RoboDK station: FollowCurves_Inatel.rdk

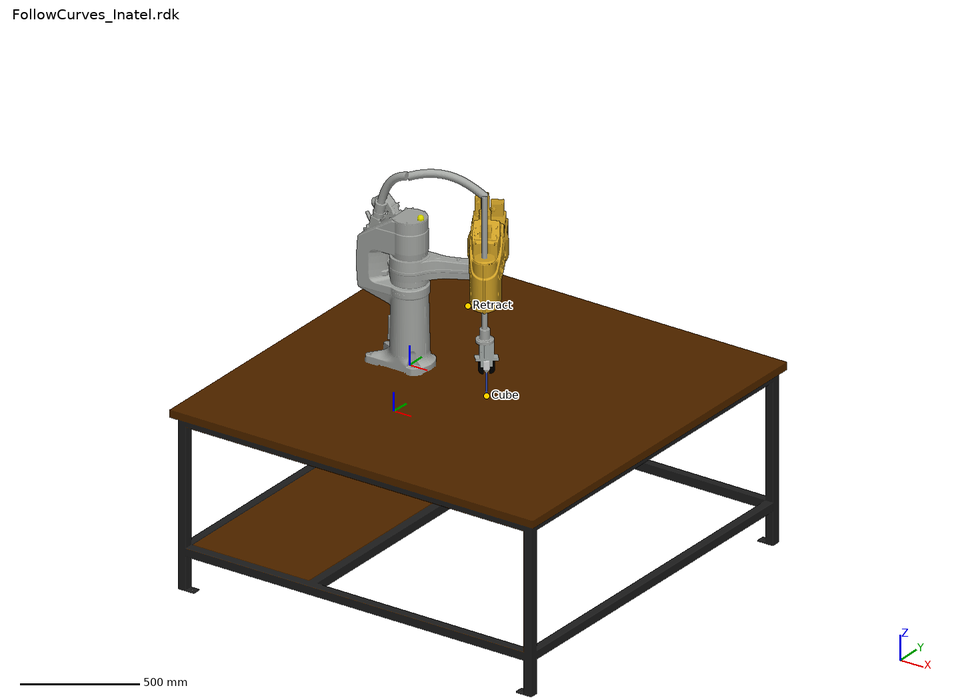
[picture v0: the station drawn from its stored meshes, robots at their saved joint values, targets as dots, program paths as lines]
Station FollowCurves_Inatel (saved by RoboDK 5.4.1). Poses are relative to the parent item; angles as X-Y-Z fixed-axis rotations.
Station parameters (name, value as stored): LIN64
  - frame World at (0, 0, 835) mm
    - robot Staubli TS60 FL 200 (model Staubli TS60 FL 400): 4 axes, payload 2 kg, reach 600 mm, repeatability 0.01 mm, weight 55 kg
        modified DH rows (alpha deg, a mm, theta deg, d mm): 0, 0, 0, 0; 0, 330, 0, 0; 0, 270, 0, 170 linear; 180, 0, 0, 0
        joint limits [-140, -150, 0, -500] to [140, 150, 200, 500]; home [0, 0, 0, 0]; saved at [27.421, -85.421, 90, 122]
      - tool GarraCompleta, TCP at (0, 0, 200) mm, size 97 x 40 x 153.1 mm, geometry from GarraCompleta.STL
        - object Suporte_e_Caneta at (4.39, 18.92, -137) mm, rotated rx 0 ry 0 rz 48 deg, size 26 x 26 x 165.9 mm, geometry from Suporte_e_Caneta.STL
      - tool TCP_Garra, TCP at (0, 17, 260) mm
    - target Retract (Cartesian target) at (-121.61, 599.78, 0) mm, rotated rx 180 ry 0 rz -180 deg; joints [108.252, -14.375, 90, 273.877] of Staubli TS60 FL 200
  - object Mesa at (350, 0, 0) mm, size 1850 x 1850 x 835 mm, geometry from Mesa.STL
  - frame AreaTrabalho at (200, -400, 835) mm
    - target Cube (Cartesian target) at (236, 340, 0) mm, rotated rx 180 ry 0 rz 180 deg; joints [22.348, -85.774, 90, 116.574] of Staubli TS60 FL 200
  - Python program dynamicTarget (listed below)

--- Python program dynamicTarget ---
from robodk.robolink import *      # RoboDK's API
from robodk.robomath import *      # Math toolbox for robots
from tkinter import *
import numpy as np
import cv2

def getElements(image):
    imgHSV = cv2.cvtColor(image, cv2.COLOR_BGR2HSV)
    lower = np.array([32, 0, 0])
    upper = np.array([145, 255, 255])
    mask = cv2.inRange(imgHSV, lower, upper)
    imgResult = cv2.bitwise_and(image, image, mask=mask)
    return imgResult

def showImages(images):
    for image in images:
        cv2.imshow('Image', image)
        cv2.waitKey(0)
        cv2.destroyAllWindows()

def getPosition():
    path = '/home/fabiofiorita/Documentos/IC-Gemeo/Localização de Objetos/DynamicTarget/bancada1.png'
    image = cv2.imread(path)
    #image = cv2.resize(image, (1200, 2000))
    maskedImage = getElements(image)

    img = maskedImage.copy()
    im_bw = cv2.cvtColor(img, cv2.COLOR_RGB2GRAY)
    #blur = cv2.GaussianBlur(im_bw, (5,5), 0)
    #im_bw = cv2.Canny(blur, 10, 90)
    contours, hierarchy = cv2.findContours(im_bw, cv2.RETR_TREE, cv2.CHAIN_APPROX_SIMPLE)
    centers = []
    for c in contours:
        M = cv2.moments(c)
        if M['m00'] != 0:
            cx = int(M['m10']/M['m00'])
            cy = int(M['m01']/M['m00'])
            cv2.drawContours(img, [c], -1, (0,255,0), 3)
            cv2.circle(img, (cx, cy), 5, (0,0,255), -1)
            cv2.putText(img, f"{cx, cy}", (cx - 20, cy - 20), cv2.FONT_HERSHEY_SIMPLEX, 0.5, (0,0,255), 2)
            centers.append((cx, cy))
    showImages([image, maskedImage, img])
    return centers

def interface():
    centers = getPosition()

    master = Tk()
    master.geometry("400x400")
    master.title("Localização de Objetos")
    master.eval('tk::PlaceWindow . center')


    t = Text(master, height=10, width=10)
    for x in centers:
        t.insert(END, x)
        t.insert(END, "\n")
    t.pack()

    indexes = []
    j = 0
    for _ in centers:
        indexes.append(j)
        j += 1

    variable = StringVar(master)
    variable.set(indexes[0])

    w = OptionMenu(master, variable, *indexes)
    w.pack()


    def ok():
        result = variable.get()
        print ("value is: " + result)
        print(centers[int(result)])
        global cx, cy
        cx, cy = centers[int(result)]
        master.destroy()

    button = Button(master, text="OK", command=ok)
    button.pack()

    mainloop()
    return cx, cy

RL = Robolink()

robot = RL.Item('Staubli TS60 FL 200')
world = RL.Item('World')
retract = RL.Item('Retract')
areaTrabalho = RL.Item('AreaTrabalho')

target = RL.AddTarget('Cube', areaTrabalho)
cx, cy = interface()
print(cx, cy)
RL.ShowMessage('Centers: ' + str(cx) + ' ' + str(cy))
target.setPose(Offset(eye(), cx, cy, 0, 0, 180, 0))

robot.MoveJ(retract)
robot.MoveJ(target)
robot.MoveJ(retract)
